FUNCTION_BLOCK FB_Gripper_GripAngle
VAR_INPUT
	lrPenDiameter	:lREAL;(*ペンの直径 単位mm*)
END_VAR
VAR_OUTPUT
	lrGripAngle		:LREAL;(*グリップする角度*)
END_VAR
VAR
	lrd				:LREAL:=6.000;(*アタッチメントの直径［mm］*)
	lrr				:LREAL:=6.400;(*アタッチメントの回転半径［mm］*)
	lrA				:LREAL;
	lrB				:LREAL;
END_VAR

	lrA:=EXPT((lrPenDiameter+lrd)/2,2)-EXPT(9.05,2)-EXPT(lrr,2);
	lrB:=2*9.05*lrr;

	IF -1<lrA/lrB AND lrA/lrB<1 THEN
		lrGripAngle:=180/PI*ACOS(lrA/lrB);
	END_IF;

END_FUNCTION_BLOCK

(* stored: Version 1.1.0.1, ProductVersion 3.1.4026.11
   POU FB_Gripper_GripAngle: Id {e4688722-634f-464e-a20f-efe8a902898e}, SpecialFunc None *)
